(* CoDeSys 2.3.9.42 project: plc.pro *)
(* Libraries: STANDARD.LIB 5.6.98 11:03:02 *)

(* Task configuration *)
TASK Standard (PRIORITY := 0, INTERVAL := T#10ms);
	MAIN
END_TASK

(* POU MAIN, ST *)
PROGRAM MAIN
VAR
	selectscreen : INT;
	bitmapdone:BOOL;
	recipewrite : BOOL;
	recipedone:BOOL;

	bmp1 : STRING(80) := 'image1.bmp';
	bmp2 : STRING(80) := 'image2.bmp';
	bmp3 : STRING(80) := 'image3.bmp';
	bmp4 : STRING(80) := 'image4.bmp';
	bmp5 : STRING(80) := 'image5.bmp';
	bmp6 : STRING(80) := 'image6.bmp';
	bmp7 : STRING(80) := 'image7.bmp';
	bmp8 : STRING(80) := 'image8.bmp';
	bmp9 : STRING(80) := 'image9.bmp';

END_VAR
;
END_PROGRAM
